FUNCTION_BLOCK StartPauseResetButtons_HMI (* Service Interface Function Block Type *)
  (* Standard: 61499-2 *)
  (* Version 0.0, 10/12/2016, Aalto_IT, nxtControl GmbH, template *)
  PACKAGE Main;
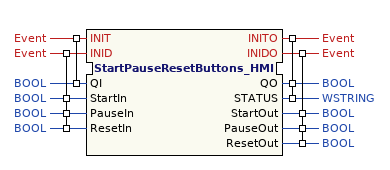
  EVENT_INPUT
    INIT WITH QI;
    INID WITH StartIn, PauseIn, ResetIn;
  END_EVENT
  EVENT_OUTPUT
    INITO WITH QO, STATUS;
    INIDO WITH StartOut, PauseOut, ResetOut;
  END_EVENT
  VAR_INPUT
    QI : BOOL;
    StartIn : BOOL;
    PauseIn : BOOL;
    ResetIn : BOOL;
  END_VAR
  VAR_OUTPUT
    QO : BOOL; (* Event Output Qualifier *)
    STATUS : WSTRING; (* Service Status *)
    StartOut : BOOL;
    PauseOut : BOOL;
    ResetOut : BOOL;
  END_VAR
END_FUNCTION_BLOCK
